FUNCTION_BLOCK AI_force
VAR_INPUT
	Raw_IO : INT;
END_VAR

VAR_OUTPUT
	Out : INT;
END_VAR

VAR
	ForceEnable : BOOL;
	ForceValue : INT;
END_VAR

IF NOT ForceEnable THEN
	OUT := Raw_IO;
ELSE
	OUT := ForceValue;
END_IF

END_FUNCTION_BLOCK

(* stored: Version 1.1.0.1, ProductVersion 3.1.4024.15
   POU AI_force: Id {8ed63623-f1d7-4795-b32d-7ddc0a6476f7}, SpecialFunc None *)
